ABB RobotStudio station: PaletizadoTPL2_final.rspag

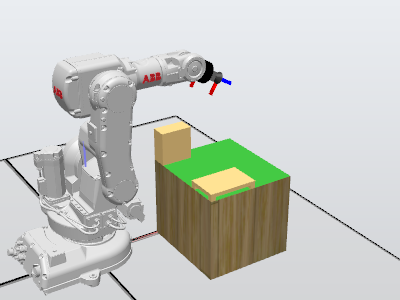
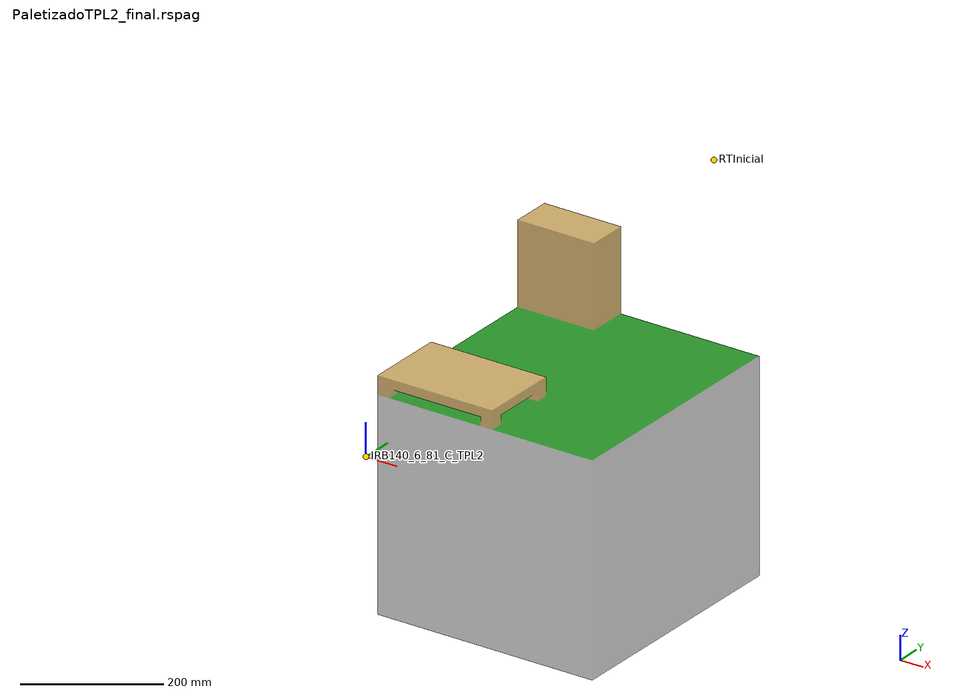
[picture v1: parts stored in the station drawn from their meshes, with robot base, taught points and paths (robot models come from the ABB library and are not in the file)]
--- station ---
Station Paletizado (saved by RobotStudio 25.3.11371.0)
Controller IRB140_6_81_TPL2
  mechanical unit ROB_1: IRB140_6_81_C_TPL2, 6 joints, base frame (0, 0, 0) mm
Layout (positions relative to the parent item):
  - Mesa [part], size 365 x 405 x 340 mm
  - Pallet [part], size 195 x 130 x 30 mm
  - Pieza1 [part], size 130 x 65 x 15 mm
  - Pieza2 [part], size 130 x 65 x 15 mm
  - Pieza3 [part], size 130 x 65 x 15 mm
  - Pieza4 [part], size 130 x 65 x 15 mm
  - Pieza5 [part], size 130 x 65 x 15 mm
  - Pieza6 [part], size 130 x 65 x 15 mm
  - Pieza7 [part], size 130 x 65 x 15 mm
  - Pieza8 [part], size 130 x 65 x 15 mm
  - Pieza9 [part], size 130 x 65 x 15 mm
  - Sopapa [mechanism] at (506.29, 0, 679.5) mm, rotated rx 180 ry 60 rz 180 deg
      TCP Sopapa at (0, -5, 103) mm
      links: Sopapa
  - IRB140_6_81_C_TPL2 [mechanism, from %ABB.RobotStudio.Models.IRB140%\IRB140_6_81_C_G_03.rslib] at (0, 0, 0) mm; joint values [0, 0, 0, 0, 0.5236, 0] (rad or m)
Attachment: Sopapa is attached to IRB140_6_81_C_TPL2 / Link6
EventTableEntry 1212: Group=, Trigger=DO_Pinza 1213, Actions=[EventTableActionAttach 1214], Comment=, ActivationMode=2, Cyclic=false
EventTableTriggerIO 1213: IOValue=[1], IRC5Controller=? -1, Operator=0, SignalSource=? -1
EventTableActionAttach 1214: AttachmentParent=Sopapa 1252, AttachmentChild=? -1, MountObject=false, Offset=[X=1, Y=0, Z=0, W=0, X=0, Y=1, Z=0, W=0, X=0, Y=0, Z=1, W=0, X=0, Y=0, Z=0, W=1], FlangeIndext=0, FindNearest=true
EventTableEntry 1219: Group=, Trigger=DO_Pinza 1220, Actions=[EventTableActionDetach 1221], Comment=, ActivationMode=2, Cyclic=false
EventTableTriggerIO 1220: IOValue=[0], IRC5Controller=? -1, Operator=0, SignalSource=? -1
EventTableActionDetach 1221: AttachmentParent=Sopapa 1252, AttachmentChild=? -1
EventTableEntry 2376: Group=, Trigger=DO_Sopapa 2377, Actions=[EventTableActionAttach 2378], Comment=, ActivationMode=2, Cyclic=false
EventTableTriggerIO 2377: IOValue=[1], IRC5Controller=? -1, Operator=0, SignalSource=IRB140_6_81_TPL2 1258
EventTableActionAttach 2378: AttachmentParent=Sopapa 1252, AttachmentChild=? -1, MountObject=false, Offset=[X=1, Y=0, Z=0, W=0, X=0, Y=1, Z=0, W=0, X=0, Y=0, Z=1, W=0, X=0, Y=0, Z=0, W=1], FlangeIndext=0, FindNearest=true
EventTableEntry 2379: Group=, Trigger=DO_Sopapa 2380, Actions=[EventTableActionDetach 2381], Comment=, ActivationMode=2, Cyclic=false
EventTableTriggerIO 2380: IOValue=[0], IRC5Controller=? -1, Operator=0, SignalSource=IRB140_6_81_TPL2 1258
EventTableActionDetach 2381: AttachmentParent=Sopapa 1252, AttachmentChild=? -1
Targets, tools, work objects and paths stored in the station and not in the controller backup, written as RAPID:
! task T_ROB1
MODULE Module1
  PROC Path_10()
    MoveL RTPosPallet3,v1000,z100,Sopapa\WObj:=WOPallet;
    MoveL RTPosPallet1,v1000,z100,Sopapa\WObj:=WOPallet;
    MoveL RTPosPallet2,v1000,z100,Sopapa\WObj:=WOPallet;
    MoveL RTCajaSuperior,v1000,z100,Sopapa\WObj:=WOCajas;
    MoveL RTInicial,v1000,z100,Sopapa\WObj:=wobj0;
  ENDPROC
ENDMODULE


--- Backups/IRB140_6_81_TPL2/RAPID/TASK1/PROGMOD/Module1.mod ---
MODULE Module1
    ! Tools
    PERS tooldata Sopapa:=[TRUE,[[0,-5,103],[1,0,0,0]],[0.5,[0,0,40],[1,0,0,0],0,0,0]];
    PERS tooldata SopapaCaja:=[TRUE,[[0,-5,118],[1,0,0,0]],[0.5,[0,0,40],[1,0,0,0],0,0,0]];

    ! Transformación de Tool
    VAR pose caja := [[0,0,15],[1,0,0,0]];

    ! WorldObjects
    TASK PERS wobjdata WOCajas:=[FALSE,TRUE,"",[[300,5,340],[0.707106781,0,0,-0.707106781]],[[0,0,0],[1,0,0,0]]];
    TASK PERS wobjdata WOPallet:=[FALSE,TRUE,"",[[300,-400,370],[1,0,0,0]],[[0,0,30],[1,0,0,0]]];

    ! RobotTargets
    CONST robtarget RTInicial:=[[595.492267836,-5,628],[0.5,0,0.866025404,0],[0,0,0,0],[9E+09,9E+09,9E+09,9E+09,9E+09,9E+09]];
    CONST robtarget RTCajaSuperior:=[[32.5,65,135],[0,-0.707106781,0.707106781,0],[-1,0,-1,0],[9E+09,9E+09,9E+09,9E+09,9E+09,9E+09]];
    CONST robtarget RTPosPallet1:=[[65,32.5,0],[0,1,0,0],[-1,0,1,0],[9E+09,9E+09,9E+09,9E+09,9E+09,9E+09]];
    CONST robtarget RTPosPallet2:=[[65,97.5,0],[0,0,1,0],[-1,0,-1,0],[9E+09,9E+09,9E+09,9E+09,9E+09,9E+09]];
    CONST robtarget RTPosPallet3:=[[162.5,65,0],[0,0.707106781,0.707106781,0],[0,0,0,0],[9E+09,9E+09,9E+09,9E+09,9E+09,9E+09]];

    ! Dimensiones Caja
    CONST num largoCaja := 130;
    CONST num anchoCaja := 65;
    CONST num altoCaja  := 15;

    ! Dimensiones Palet
    CONST num largoPalet := 195;
    CONST num anchoPalet := 130;

    ! Parámetros
    CONST num N_Cajas := 9;
    CONST num CajasPorPiso := 3;
    CONST robtarget posiciones{3} := [RTPosPallet1, RTPosPallet2, RTPosPallet3];
    CONST num posOffs{3,2} := [[-1,-1], [-1,1], [1,0]];

    ! Distancia para acercarse/alejarse con MoveJ
    CONST num offset := 20;

    ! Variables
    VAR num CajasEnPalet;
    VAR num Piso;
    VAR num aux;

    PROC main()
        MoveJ RTInicial,v100,fine,Sopapa\WObj:=wobj0;
        Reset DO_Sopapa;
        WOPallet.oframe := [[0,0,0],[1,0,0,0]];

        CajasEnPalet := 0;
        aux := CajasEnPalet MOD CajasPorPiso;
        piso := 1 + (CajasEnPalet DIV CajasPorPiso);


        WHILE CajasEnPalet < N_Cajas DO
            IF piso MOD 2 = 0 THEN
                WOPallet.oframe := [[largoPalet, anchoPalet, (piso-1)*altoCaja],[0,0,0,1]];
            ELSE
                WOPallet.oframe := [[0, 0, (piso-1)*altoCaja],[1,0,0,0]];
            ENDIF

            FOR j FROM aux+1 TO 3 DO
                Pick CajasEnPalet;
                Place posiciones{j}, posOffs{j,1}, posOffs{j,2};
                CajasEnPalet := CajasEnPalet + 1;
            ENDFOR
            aux := 0;
            Piso := Piso + 1;
        ENDWHILE
        MoveJ RTInicial,v100,fine,Sopapa\WObj:=wobj0;

    ENDPROC

    PROC Pick(num nCajasAgarradas)
        MoveJ Offs(RTCajaSuperior,0,0,-nCajasAgarradas*altoCaja + offset),v100,z50,Sopapa\WObj:=WOCajas;
        MoveL Offs(RTCajaSuperior,0,0,-nCajasAgarradas*altoCaja),v100,fine,Sopapa\WObj:=WOCajas;
        WaitTime 1;
        Set DO_Sopapa;
        WaitTime 1;
        SopapaCaja.tframe := PoseMult(Sopapa.tframe, caja);
        MoveL Offs(RTCajaSuperior,0,0,-nCajasAgarradas*altoCaja + offset),v100,fine,SopapaCaja\WObj:=WOCajas;
    ENDPROC

    PROC Place(robtarget destino, num offs_x, num offs_y)
        MoveJ Offs(destino, offs_x*offset, offs_y*offset, offset),v100,z100,SopapaCaja\WObj:=WOPallet;
        MoveL destino,v50,fine,SopapaCaja\WObj:=WOPallet;
        WaitTime 1;
        Reset DO_Sopapa;
        WaitTime 1;
        MoveL Offs(destino,0,0,offset),v100,fine,Sopapa\WObj:=WOPallet;
    ENDPROC

ENDMODULE

--- Backups/IRB140_6_81_TPL2/SYSPAR/EIO.cfg ---
EIO:CFG_1.0:6:1::
#
EIO_SIGNAL:

      -Name "DO_Sopapa" -SignalType "DO" -Access "All"
